// TwinCAT 3 PLC project plc01
// ProgramVersion: 3.1.4026.19
// libraries:
//   Tc2_Standard, * (Beckhoff Automation GmbH)
//   Tc2_System, * (Beckhoff Automation GmbH)
//   Tc2_Utilities, * (Beckhoff Automation GmbH)
//   Tc3_EventLogger, * (Beckhoff Automation GmbH)
//   Tc3_JsonXml, * (Beckhoff Automation GmbH)
//   [Tc3_Logging], * (www.peterzerlauth.com)
// project tree:
//   / FastTask.TcTTO (not stored), PlcTask.TcTTO (not stored)
//   POUs/ FAST.TcPOU, MAIN.TcPOU
//   POUs/FileLogging/ FB_FileLogging.TcPOU (not stored)
//   POUs/File/ E_File.TcDUT, FB_File.TcPOU
//   POUs/LinkedList/ FB_LoggerList.TcPOU, ST_LoggingNode.TcDUT (not stored)
//   POUs/TcAlarming/ FB_TcAlarming.TcPOU (not stored)
// real-time tasks:
//   TASK SlowTask: cycle T#20ms, priority 20, ADS port 350
//   TASK FastTask: cycle T#1ms, priority 1, ADS port 351

// ---- POUs/File/E_File.TcDUT
{attribute 'qualified_only'}
{attribute 'strict'}
{attribute 'to_string'}
TYPE E_File :
(
	Idle		:= 0,
	Info		:= 1,
	Create		:= 2,
	Open		:= 9,
	Read		:= 10,
	Write		:= 11,
	Close		:= 12
);
END_TYPE

// ---- POUs/FAST.TcPOU
PROGRAM FAST
VAR
	fbLogger:			FB_Logger;
	bVerbose:			BOOL;
	bInfo:				BOOL;
	bWarning:			BOOL;
	bError:				BOOL;
	bCritical:			BOOL;
END_VAR

fbLogger.P_Logger:= MAIN.fbLogging;

IF bVerbose THEN
	fbLogger.P_Argument.M_AddINT(134052566194980000);
	fbLogger.P_Argument.M_AddSTRING('mm');
	fbLogger.M_Verbose('Verbose message %s %s');
END_IF

IF bInfo THEN
	fbLogger.M_Info(2276475569, 'Info message');END_IF

IF bWarning THEN

	fbLogger.M_Info(2276475569, 'Info message');
	fbLogger.M_Warning(1791326186, 'Warning message');
	fbLogger.M_Error(2621541999, 'Error message');
END_IF

IF bError THEN
	fbLogger.M_Info(2276475569, 'Info message');
END_IF

IF bCritical THEN
	fbLogger.M_Critical(2626343866, 'Critical message');
END_IF

END_PROGRAM

// ---- POUs/MAIN.TcPOU
PROGRAM MAIN
VAR
// 	fbLoggerList:		FB_LoggerList;
// 	fbFile:				FB_File;
	fbLogging:			FB_Logging;
	fbTcLogging:		FB_TcLogging;
	fbTcAlarming:		FB_TcAlarming;
	fbLogger:			FB_Logger;
	bVerbose:			BOOL;
	bInfo:				BOOL;
	bWarning:			BOOL;
	bError:				BOOL;
	bCritical:			BOOL;
	bOpen: 				BOOL;
END_VAR

// fbFile();
// IF bOpen THEN
// 	bOpen:= NOT fbFile.M_Open('C:\temp\log.txt');
// END_IF

fbLogging();
fbLogging.M_Attach(fbTcLogging);

fbTcLogging();

fbTcAlarming();

fbLogger.iLogging:= fbLogging;

fbLogger();

// fbLoggerList.M_Add(fbTcLogging);



IF bVerbose THEN
	fbLogger.P_Argument.M_AddINT(134052566194980000);
	fbLogger.P_Argument.M_AddSTRING('mm');
	fbLogger.M_Verbose('message %s %s');
END_IF

IF bInfo THEN
	fbLogger.P_Argument.M_AddREAL(33.134581234, 3);
	fbLogger.P_Argument.M_AddSTRING('mm');
	fbLogger.M_Info(2263151477, 'message %s %s');
END_IF

IF bWarning THEN
	fbLogger.M_Warning(292272521, 'message');
END_IF

IF bError THEN
	fbLogger.M_Error(292272521, 'message');
END_IF

IF bCritical THEN
	fbLogger.M_Critical(292272521, 'message');
END_IF

END_PROGRAM

// ---- POUs/File/FB_File.TcPOU
FUNCTION_BLOCK FB_File
VAR
	fbInfo:			 	FB_FileProperties;
    fbCreateDir:		FB_CreateDir;
	fbOpen:				FB_FileOpen;
	fbRead:				FB_FileRead;
	fbWrite:			FB_FileWrite;
	fbClose:			FB_FileClose;
	fbDelete:			FB_FileDelete; 
END_VAR
VAR_OUTPUT
	bBusy:					BOOL;
	bError:					BOOL;
	nErrId:					UDINT;
END_VAR
VAR CONSTANT
	nMaxFileSize:		UDINT:= 1024 * 1024;
END_VAR

fbInfo();
fbCreateDir();
fbOpen();
fbRead();
fbWrite();
fbClose();
fbDelete();

METHOD PUBLIC M_Append : BOOL
VAR_INPUT
	Text:			STRING(255);
END_VAR
IF fbWrite.bExecute THEN
	IF fbWrite.bError THEN
		nErrId:= fbWrite.nErrId;
		fbWrite.bExecute:= FALSE;
	ELSIF fbWrite.bBusy THEN
		;
	ELSE
		M_Append:= TRUE;
		fbWrite.bExecute:= FALSE;
	END_IF
ELSE
	fbWrite.bExecute:= TRUE;
	fbWrite.pWriteBuff:= ADR(Text);
	fbWrite.cbWriteLen:= INT_TO_UDINT(Len(Text));
END_IF
END_METHOD

METHOD PUBLIC M_Close : BOOL
VAR_INPUT
END_VAR
IF fbClose.bExecute THEN
	IF fbClose.hFile = 0 THEN
		fbClose.bExecute:= FALSE;
		M_Close:= TRUE;
	ELSIF fbClose.bError THEN
		fbClose.bExecute:= FALSE;
		nErrId:= fbClose.nErrId;
	ELSIF fbClose.bBusy THEN
		;
	ELSE
		nErrId:= 0;	
		fbRead.hFile:= 0;
		fbWrite.hFile:= 0;
		fbClose.hFile:= 0;
		fbClose.bExecute:= FALSE;
		M_Close:= TRUE;
	END_IF
ELSE
	fbClose.bExecute:= TRUE;
END_IF
END_METHOD

METHOD PUBLIC M_Create : BOOL
VAR_INPUT
	sPathName:		STRING(255);
END_VAR
VAR
	nTemp: INT;
END_VAR
VAR_INST
	nPosition: INT;
END_VAR
nTemp := FIND(RIGHT(sPathName, LEN(sPathName) - nPosition), '\');
if nTemp <> 0 then
	IF fbCreateDir.bExecute THEN
		IF NOT fbCreateDir.bBusy THEN
			nPosition := nPosition + nTemp;
			fbCreateDir.bExecute:= FALSE;
		END_IF
	ELSE
		fbCreateDir.bExecute:= TRUE;
		fbCreateDir.ePath:= PATH_GENERIC;
		fbCreateDir.sPathName:= Left(sPathName, nPosition + nTemp);
	END_IF
ELSE
	M_Create:= TRUE;
END_IF
END_METHOD

METHOD PUBLIC M_Delete : BOOL
VAR_INPUT
	PathName:		STRING(255);
END_VAR
fbDelete();
IF fbDelete.bExecute THEN
	IF fbDelete.bError THEN
		fbDelete.bExecute:= FALSE;
		M_Delete:= TRUE;
	ELSIF fbDelete.bBusy THEN
		;
	ELSE
		fbDelete.bExecute:= FALSE;
		M_Delete:= TRUE;
	END_IF
ELSE
	fbDelete.bExecute:= TRUE;
	fbDelete.sPathName:= PathName;
	fbDelete.ePath:= E_OpenPath.PATH_GENERIC;
END_IF
END_METHOD

METHOD PUBLIC M_Open : BOOL
VAR_INPUT
	sPathName:		STRING(255);
END_VAR
IF fbOpen.bExecute THEN
	IF fbOpen.bError THEN
		nErrId:= fbOpen.nErrId;
		fbOpen.bExecute:= FALSE;
	ELSIF fbOpen.bBusy THEN
		;
	ELSE
		fbRead.hFile:= fbOpen.hFile;
		fbWrite.hFile:= fbOpen.hFile;
		fbClose.hFile:= fbOpen.hFile;
		fbOpen.bExecute:= FALSE;
		M_Open:= TRUE;
	END_IF	
ELSE
	IF M_Create(sPathName) THEN
		fbOpen.bExecute:= TRUE;
		fbOpen.sPathName:= sPathName;
		fbOpen.nMode:= (FOPEN_MODEAPPEND OR FOPEN_MODEPLUS OR FOPEN_MODETEXT);		
	END_IF
END_IF
END_METHOD

METHOD PUBLIC M_Read : BOOL
VAR_INPUT
	Value:		ANY;
END_VAR
IF fbRead.bExecute THEN
	IF fbRead.bError THEN
		nErrId:= fbRead.nErrId;
		fbRead.bExecute:= FALSE;
	ELSIF fbRead.bBusy THEN
		;
	ELSE
		fbRead.bExecute:= FALSE;
		M_Read:= TRUE;
	END_IF
ELSE
	fbRead.bExecute:= TRUE;
END_IF
END_METHOD

METHOD PUBLIC M_Write : BOOL
VAR_INPUT
	Value:		ANY;
END_VAR
IF fbWrite.bExecute THEN
	IF fbWrite.bError THEN
		nErrId:= fbWrite.nErrId;
		fbWrite.bExecute:= FALSE;
	ELSIF fbWrite.bBusy THEN
		M_Write:= FALSE;
	ELSE
		M_Write:= TRUE;
		fbWrite.bExecute:= FALSE;
	END_IF
ELSE
	fbWrite.bExecute:= TRUE;
END_IF
END_METHOD

END_FUNCTION_BLOCK

// ---- POUs/LinkedList/FB_LoggerList.TcPOU
FUNCTION_BLOCK FB_LoggerList IMPLEMENTS I_Logging
VAR_INPUT
END_VAR
VAR_OUTPUT
END_VAR
VAR
	pLoggingNode: 	POINTER TO St_LoggingNode;
END_VAR

METHOD PUBLIC M_Add : BOOL
VAR_INPUT
	iLogging:  I_Logging;
END_VAR
VAR
	pNewNode : POINTER TO St_LoggingNode;
	pIter    : POINTER TO St_LoggingNode;
END_VAR
// Allocate new node
pNewNode := __NEW(ST_LoggingNode);
IF pNewNode = 0 THEN 
	RETURN;
END_IF

// Assign interface pointer
pNewNode^.pLogger := iLogging;
pNewNode^.pNext := 0;

// Append to list
IF pLoggingNode = 0 THEN
	pLoggingNode := pNewNode;
ELSE
	pIter := pLoggingNode;
	WHILE pIter^.pNext <> 0 DO
		pIter := pIter^.pNext;
	END_WHILE
	pIter^.pNext := pNewNode;
END_IF

M_Add := TRUE;
END_METHOD

METHOD PUBLIC M_Delete : BOOL
VAR_INPUT
END_VAR
VAR
	pIter, pNext : POINTER TO St_LoggingNode;
END_VAR
pIter := pLoggingNode;
WHILE pIter <> 0 DO
	pNext := pIter^.pNext;
	__DELETE(pIter);
	pIter := pNext;
END_WHILE
pLoggingNode := 0;
M_Delete:= TRUE;
END_METHOD

METHOD M_Log : BOOL
VAR_INPUT
	stMessage	: Tc3_Logging.ST_Message;
END_VAR
VAR
	pIter : POINTER TO St_LoggingNode;
END_VAR
pIter := pLoggingNode;
WHILE pIter <> 0 DO
	IF pIter^.pLogger <> 0 THEN
		pIter^.pLogger^.M_Log(stMessage);
	END_IF
	pIter := pIter^.pNext;
END_WHILE
M_Log:= TRUE;
END_METHOD

END_FUNCTION_BLOCK
